// TIA Portal V20 export
// export: Created 2025-09-12T17:59:00.0000000Z, ExportSetting WithDefaults
FUNCTION_BLOCK "FB300_EM_Heating"   // FB, SCL
TITLE = EM-300: Heating Control
AUTHOR : Dallas Levine
VERSION : 0.1
// This block contains all logic for the Heating Equipment Module (EM-300).
// stored: AutoNumber true, IsRetain false
   VAR_INPUT
      Enable : Bool;   // Enables the block's execution.
      Valve_Demand_In : Real;   // Demand signal from the main PID controller (0.0 - 100.0 %).
   END_VAR
   VAR
      UDT : "UDT300_EM_Heating";   // The data interface for the Heating Equipment Module.
      Feedback_Fault_Timer : TON_TIME;   // Timer for the feedback fault delay.
   END_VAR
   VAR CONSTANT
      FEEDBACK_TOLERANCE : Real := 10.0;   // Allowable deviation between command and feedback (%).
      FEEDBACK_DELAY : Time := T#60s;   // Time delay before a feedback mismatch becomes an alarm.
   END_VAR
BEGIN
   REGION Main Logic 
   IF #Enable THEN

    (/**/) #UDT.HW_Valve_Cmd_AO := #Valve_Demand_In;

    (/**/) #UDT.HW_Freeze_Alm := #UDT.HW_Freeze_Stat_DI;
    IF #UDT.HW_Freeze_Alm THEN
     #UDT.HW_Valve_Cmd_AO := 0.0;
    END_IF;

    (/**/) #Feedback_Fault_Timer(IN:= ABS(FV:=#UDT.HW_Valve_Cmd_AO - #UDT.HW_Valve_Fdbk_AI) > #FEEDBACK_TOLERANCE,
           PT:= #FEEDBACK_DELAY);
    #UDT.Valve_Failure_Alm := #Feedback_Fault_Timer.Q;
   ELSE
    (/**/) #UDT.HW_Valve_Cmd_AO := 0.0;
    #UDT.Valve_Failure_Alm := FALSE;
   END_IF;
   END_REGION
END_FUNCTION_BLOCK
